{attribute 'qualified_only'}
VAR_GLOBAL
END_VAR

(* stored: Version 1.1.0.1, ProductVersion 3.1.4022.12
   GVL GVL_TimeConstants: Id {2cbdfe05-3b59-43e7-8e60-9be230e93c32} *)
